// Returns TRUE if possible. sVal will hold value if passes. 
//
// Internally this casts to Udint, then checks value is <= MAX_WORD
FUNCTION TryStringToWord : BOOL
VAR_INPUT
   sStringToParse : STRING; // String to try
END_VAR
VAR_IN_OUT
   sVal : WORD; // 0 (zero) if fails, parsed value if passes.
END_VAR
VAR
   u : UDINT;
END_VAR

// check parsing to UDINT possible, then validate size of word.
IF TryStringToUdint(sStringToParse, u) THEN
   // check within WORD size.
   IF UDINT_TO_WORD(u) <= 65535 THEN
      sVal := STRING_TO_WORD(sStringToParse);
      TryStringToWord := TRUE;
   END_IF

END_IF

END_FUNCTION

(* stored: Version 1.1.0.1, ProductVersion 3.1.4024.9
   POU TryStringToWord: Id {f01d99cf-ccb1-4a2a-aebc-0259bb8a74f4}, SpecialFunc None *)
